RoboDK station: _.rdk

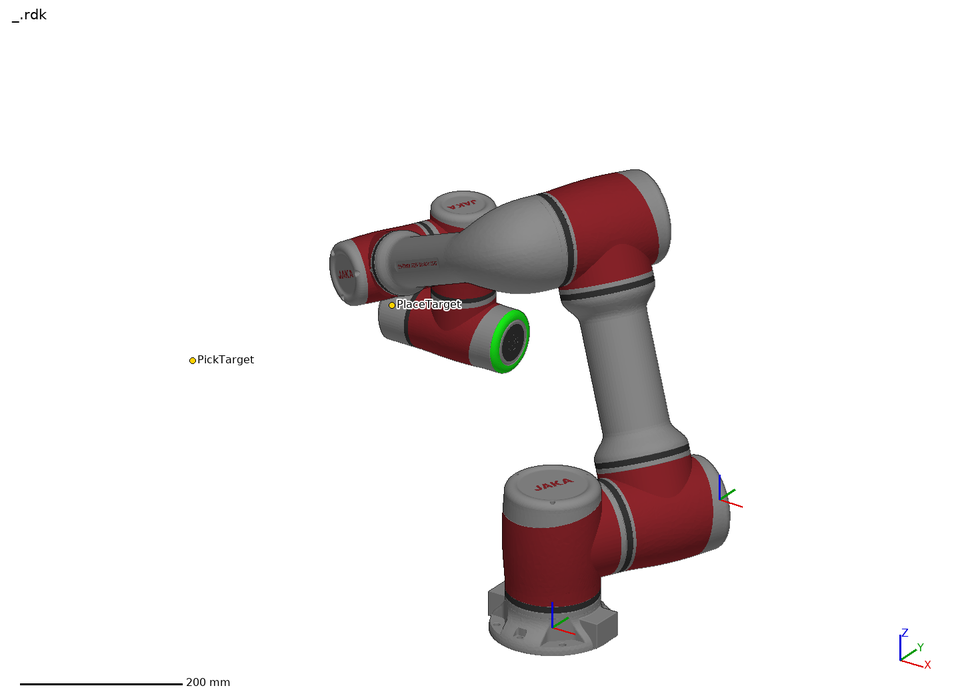
[picture v0: the station drawn from its stored meshes, robots at their saved joint values, targets as dots, program paths as lines]
Station  (saved by RoboDK 5.9.1). Poses are relative to the parent item; angles as X-Y-Z fixed-axis rotations.
  - frame JAKA Zu7 at (0, 0, 0) mm
    - robot JAKA Zu7: 6 axes
        modified DH rows (alpha deg, a mm, theta deg, d mm): 0, 0, 0, 120.15; 90, 0, 0, 0; 0, 360, 0, 0; 0, 303.5, -180, -115.01; -90, 0, 0, 113.5; 90, 0, 0, 107
        joint limits [-360, -85, -175, -85, -360, -360] to [360, 265, 175, 265, 360, 360]; home [0, 90, 90, 180, 90, 0]; saved at [-25.043, 113.882, 91.536, 154.582, 64.957, 0]
  - frame Frame 2 at (0, 358.19, 31.6) mm
    - target PlaceTarget (Cartesian target) at (-438.71, -76.26, 173.96) mm, rotated rx 90 ry 0 rz -90 deg; joints [32.697, 102.665, 114.638, 142.698, 122.697, 0] of JAKA Zu7
    - target PickTarget (Cartesian target) at (-534.75, -366.76, 187.71) mm, rotated rx 90 ry 0 rz -90 deg; joints [165.554, 43.663, -103.683, 240.02, 104.446, -180] of JAKA Zu7
